Universal Robots PolyScope program: Gripper_UR_Control.urp

Program Gripper_UR_Control (installation=default directory=/programs/usbdisk createdIn=5.11.6.1010389 lastSavedIn=5.11.6.1010389 robotSerialNumber=20215301233)
Calibrated DH parameters: a=[-0.000117, -0.236381, -0.195992, 0.000035, -0.000038, 0]; d=[0.151963, 11.789192, 17.53153, -29.189907, 0.085384, 0.092292]; alpha=[1.572476, -0.005072, 0.002889, 1.571659, -1.572595, 0]; deltaTheta=[0, -0.247766, 6.938923, -0.407974, 0.000016, 0]
Robot Program (runOnlyOnce=false)
  gr_open := gripperopen
  gr_close := gripperclose
  If gr_open
    URCap Gripper Move (ROBOTIS Gripper (RH-P12-RN), ROBOTIS Co.,Ltd.) dataModel(WaitForMove=true, Current=60)
  If gr_close
    URCap Gripper Move (ROBOTIS Gripper (RH-P12-RN), ROBOTIS Co.,Ltd.) dataModel(Position=0, Current=60, WaitForMove=true)
  Wait Sleep waitTime=0.01
  If xdown
    MoveL speed 150 mm/s, acceleration 1200 mm/s^2 (useActiveTCP=true) feature=Base
      MoveDirectionNode (selectedDirection=XMinus)
        Until DISTANCE (allowActions=false deceleration=3 distanceNodeType=STOP) Distance=0.002; motionParameters(blendRadius=0)
  If xup
    MoveL speed 150 mm/s, acceleration 1200 mm/s^2 (useActiveTCP=true) feature=Base
      MoveDirectionNode (selectedDirection=XPlus)
        Until DISTANCE (allowActions=false deceleration=3 distanceNodeType=STOP) Distance=0.002; motionParameters(blendRadius=0)
  If ydown
    MoveL speed 150 mm/s, acceleration 1200 mm/s^2 (useActiveTCP=true) feature=Base
      MoveDirectionNode (selectedDirection=YMinus)
        Until DISTANCE (allowActions=false deceleration=3 distanceNodeType=STOP) Distance=0.002; motionParameters(blendRadius=0)
  If yup
    MoveL speed 150 mm/s, acceleration 1200 mm/s^2 (useActiveTCP=true) feature=Base
      MoveDirectionNode (selectedDirection=YPlus)
        Until DISTANCE (allowActions=false deceleration=3 distanceNodeType=STOP) Distance=0.002; motionParameters(blendRadius=0)
  If zdown
    MoveL speed 150 mm/s, acceleration 1200 mm/s^2 (useActiveTCP=true) feature=Base
      MoveDirectionNode (selectedDirection=ZMinus)
        Until DISTANCE (allowActions=false deceleration=3 distanceNodeType=STOP) Distance=0.002; motionParameters(blendRadius=0)
  If zup
    MoveL speed 150 mm/s, acceleration 1200 mm/s^2 (useActiveTCP=true) feature=Base
      MoveDirectionNode (selectedDirection=ZPlus)
        Until DISTANCE (allowActions=false deceleration=3 distanceNodeType=STOP) Distance=0.002; motionParameters(blendRadius=0)
